{attribute 'GeneratedUsingTerminal: ATH2040-5250-0022'}
{attribute addProperty BoxType "ATH2040-5250-0022"}
{attribute addProperty Id "BinaryDataAT %I*ARRAY [0..59] OF BYTE0"}
{attribute addProperty CRC "29753413"}
{attribute addProperty Size "0"}
TYPE FB_Inputs_01C60045 :
STRUCT
	{attribute addProperty Name "BinaryData"}
	BinaryData AT %I* : ARRAY [0..59] OF BYTE;
END_STRUCT
END_TYPE

(* stored: Version 1.2.0.0, ProductVersion 3.1.4024.9
   DUT FB_Inputs_01C60045: Id {055044ae-ad5c-4863-bc94-508c5ec06169} *)
